ORGANIZATION_BLOCK "TimeErrorInterrupt"   // OB80, LAD, TimeErrorInterrupt
{ S7_Optimized_Access := 'TRUE' }
// stored: SetENOAutomatically false
   VAR_INPUT
      Fault_ID : Byte;   // Fault identifier
      Csg_OBnr : OB_ANY;   // Number of OB causing the error
      Csg_Prio : UInt;   // Priority of OB causing the error
   END_VAR
BEGIN
END_ORGANIZATION_BLOCK

DATA_BLOCK "Instace_FB_Search_Water_Foutain_DB"   // DB109
// stored: AutoNumber false, InstanceOfName FB_Search_Water_Foutain, InstanceOfType FB
"FB_Search_Water_Foutain"
BEGIN
END_DATA_BLOCK

DATA_BLOCK "Instance_FB_DataLog_DB"   // DB110
// stored: AutoNumber false, InstanceOfName FB_DataLog, InstanceOfType FB
"FB_DataLog"
BEGIN
END_DATA_BLOCK

DATA_BLOCK "Instance_FB_Digita_Inputs_DB"   // DB101
// stored: AutoNumber false, InstanceOfName FB_Digita_Inputs, InstanceOfType FB
"FB_Digita_Inputs"
BEGIN
END_DATA_BLOCK

DATA_BLOCK "Instance_FB_Digital_Outputs_DB"   // DB103
// stored: AutoNumber false, InstanceOfName FB_Digital_Outputs, InstanceOfType FB
"FB_Digital_Outputs"
BEGIN
END_DATA_BLOCK

DATA_BLOCK "Instance_FB_HMI_DB"   // DB111
// stored: AutoNumber false, InstanceOfName FB_HMI, InstanceOfType FB
"FB_HMI"
BEGIN
END_DATA_BLOCK

DATA_BLOCK "Instance_FB_IO_Device_Functional_Test_DB"   // DB104
// stored: AutoNumber false, InstanceOfName FB_IO_Device_Functional_Test, InstanceOfType FB
"FB_IO_Device_Functional_Test"
BEGIN
END_DATA_BLOCK

DATA_BLOCK "Instance_FB_IO_Device_Functional_Test_Rework_DB"   // DB112
// stored: AutoNumber false, InstanceOfName FB_IO_Device_Functional_Test_Rework, InstanceOfType FB
"FB_IO_Device_Functional_Test_Rework"
BEGIN
END_DATA_BLOCK

DATA_BLOCK "Instance_FB_IO_Device_Production_And_Rework_DB"   // DB105
// stored: AutoNumber false, InstanceOfName FB_IO_Device_Production_And_Rework, InstanceOfType FB
"FB_IO_Device_Production_And_Rework"
BEGIN
END_DATA_BLOCK

DATA_BLOCK "Instance_FB_Marrige_DB"   // DB108
// stored: AutoNumber false, InstanceOfName FB_Marrige, InstanceOfType FB
"FB_Marrige"
BEGIN
END_DATA_BLOCK

DATA_BLOCK "Instance_FB_Read_Data_SR-X100W_Entrace_DB"   // DB106
// stored: AutoNumber false, InstanceOfName FB_Read_Data_SR-X100W, InstanceOfType FB
"FB_Read_Data_SR-X100W"
BEGIN
END_DATA_BLOCK

DATA_BLOCK "Instance_FB_Read_Data_SR-X100W_Exit_DB"   // DB107
// stored: AutoNumber false, InstanceOfName FB_Read_Data_SR-X100W, InstanceOfType FB
"FB_Read_Data_SR-X100W"
BEGIN
END_DATA_BLOCK
